// TIA Portal V20 export
FUNCTION_BLOCK "FB_Impulsion"   // FB52, SCL
{ S7_Optimized_Access := 'TRUE' }
// stored: MemoryReserve 100, SetENOAutomatically false
   VAR RETAIN
      sCountSecPulseMinute : DInt;
      sCountSecPulseHour : DInt;
      sCountSecPulseDay : DInt;
   END_VAR
   VAR
      sPulseMinute : Bool;   // Impulsion every minute
      sPulseHour : Bool;   // Impulsion every hour
      sPulseDay : Bool;   // Impulsion every day
      sRT_Clock_1Hz { S7_SetPoint := 'True'} : R_TRIG;
   END_VAR
   VAR CONSTANT
      MAX_COUNT_MINUTE : DInt := 60;
      MAX_COUNT_HOUR : DInt := 3600;
      MAX_COUNT_DAY : DInt := 86400;
   END_VAR
BEGIN
   REGION Description header 
       //==================================================================================
       // POSALUX Swiss SA / (C) Copyright 2024
       //----------------------------------------------------------------------------------
       // Title: Time counter
       // Comment/Function: Generates periodic pulses using 1Hz clock base
       //                      - Minute interval pulses (60s cycle)
       //                      - Hour interval pulses (3600s cycle)
       //                      - Day interval pulses (86400s cycle)
       //                   Implementation: Uses cascaded counters with 1Hz clock input
       // Author: Gowsigan SRITHARAN
       // Engineering: TIA Portal v17
       //----------------------------------------------------------------------------------
       // Change log table:
       // Version  | Date     | Expert in charge | Changes applied
       // ---------|----------|------------------|------------------------------------
       // 00.00.01 | 20241206 | GSR              | First released version
       // ---------|----------|------------------|------------------------------------
       // 01.01.01 | 20241219 | FMI              | Utilisation d'un flanc montant du clock1Hz pour compter en secondes
       // ==================================================================================
   END_REGION

   REGION Rising edge detection and counter incrementation
       #sRT_Clock_1Hz.CLK:="Clock_1Hz";
       #sRT_Clock_1Hz();
     IF  #sRT_Clock_1Hz.Q THEN
       #sCountSecPulseMinute := #sCountSecPulseMinute + 1;
       #sCountSecPulseHour := #sCountSecPulseHour + 1;
       #sCountSecPulseDay := #sCountSecPulseDay + 1;
   END_IF;
   END_REGION

   REGION Pulse generation and counter reset
       // Impulsion minute
       IF #sCountSecPulseMinute >= #MAX_COUNT_MINUTE THEN
           #sPulseMinute := TRUE;
           #sCountSecPulseMinute := 0;
       ELSE
           #sPulseMinute := FALSE;
       END_IF;

       // Impulsion hour
       IF #sCountSecPulseHour >= #MAX_COUNT_HOUR THEN
           #sPulseHour := TRUE;
           #sCountSecPulseHour := 0;
       ELSE
           #sPulseHour := FALSE;
       END_IF;

       // Impulsion day
       IF #sCountSecPulseDay >= #MAX_COUNT_DAY THEN
           #sPulseDay := TRUE;
           #sCountSecPulseDay := 0;
       ELSE
           #sPulseDay := FALSE;
       END_IF;
   END_REGION
END_FUNCTION_BLOCK
